TYPE EL3052_CHANNEL :
	STRUCT
		
	
	Status 	AT %I* : EL3052_DEV_STATUS;
	Value 	AT %I* : INT;
	
	
	END_STRUCT
END_TYPE

(* stored: Version 1.1.0.1, ProductVersion 3.1.4024.15
   DUT EL3052_CHANNEL: Id {574a751a-91c2-41cd-8923-960a8aff737f} *)
